// TIA Portal V16 program export: 1 tag tables, 0 data types, 0 data blocks, 3 code blocks (in call order from the OBs), 1 instance data blocks

VAR_GLOBAL   // PLC tag table "Default tag table"
   Tag_1 AT %M0.0 : Bool;
   Tag_2 AT %M10.0 : Bool;
END_VAR

ORGANIZATION_BLOCK "Main"   // OB1, LAD, ProgramCycle
TITLE = "Main Program Sweep (Cycle)"
{ S7_Optimized_Access := 'TRUE' }
VERSION : 0.1
// stored: AutoNumber true, IsIECCheckEnabled false, SetENOAutomatically false
   VAR_INPUT
      Initial_Call : Bool;   // Initial call of this OB
      Remanence : Bool;   // =True, if remanent data are available
   END_VAR
BEGIN

REGION Network 1
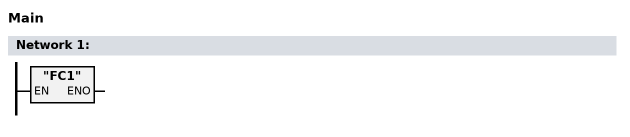
   RUNG wire#powerrail
      "FC1"()
   END_RUNG
   // the same network as SCL:
   "FC1"();
END_REGION
END_ORGANIZATION_BLOCK

FUNCTION "FC1" : Void   // FC1, LAD
{ S7_Optimized_Access := 'TRUE' }
VERSION : 0.1
// stored: AutoNumber true, IsIECCheckEnabled false, SetENOAutomatically false, UDAEnableTagReadback false
BEGIN

REGION Network 1
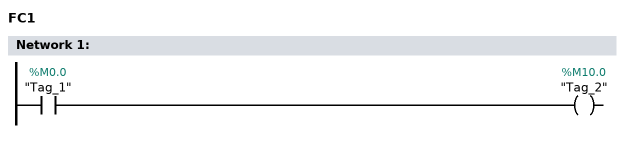
   RUNG wire#powerrail
      Contact( "Tag_1" )
      Coil( "Tag_2" )
   END_RUNG
   // the same network as SCL:
   "Tag_2" := "Tag_1";
END_REGION
END_FUNCTION

FUNCTION_BLOCK "FB1"   // FB1, LAD
{ S7_Optimized_Access := 'TRUE' }
VERSION : 0.1
// stored: AutoNumber true, IsIECCheckEnabled false, IsRetainMemResEnabled false, MemoryReserve 100, SetENOAutomatically false, UDAEnableTagReadback false
BEGIN

REGION Network 1
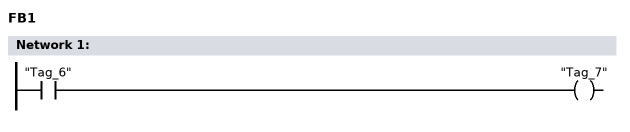
   RUNG wire#powerrail
      Contact( "Tag_6" )
      Coil( "Tag_7" )
   END_RUNG
   // the same network as SCL:
   "Tag_7" := "Tag_6";
END_REGION
END_FUNCTION_BLOCK

DATA_BLOCK "FB1_DB"   // DB1
VERSION : 0.1
// stored: AutoNumber true, DBAccessibleFromOPCUA true, InstanceOfName FB1, InstanceOfType FB
"FB1"
BEGIN
END_DATA_BLOCK
